FUNCTION_BLOCK fbEM
VAR_IN_OUT
	em : ST_EM;     
	un : ST_UN;     
END_VAR
VAR
	emCmdOld: E_CMD;
END_VAR

// Empty for now universal basic em class, every module needs to extends this to ensure compatibility

END_FUNCTION_BLOCK

(* stored: Version 1.1.0.1, ProductVersion 3.1.4024.12
   POU fbEM: Id {20ab5818-6755-4885-a642-a71cb67ceff3}, SpecialFunc None *)
